SUBAPPLICATION LinksRechts_T_FF_Event (* Links/Rechts Umschaltung mittels Toggle-Flip-Flop (E_T_FF, Event/BOOL-basiert, keine Adapter). Schwester-Baustein zu MyLib::sys::AX_LinksRechts_T_FF (dort AX-Adapter-basiert). *)
  (* Standard: 61499-2 *)
  (* Version 1.0, 2026-09-09, Franz Höpfinger, Meisterschulen am Ostbahnhof, Ausgelagert aus Uebung_006a3_sub zur Wiederverwendung. *)
  PACKAGE MyLib::sys;
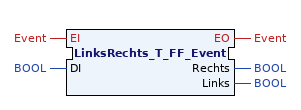
  EVENT_INPUT
    EI;
  END_EVENT
  EVENT_OUTPUT
    EO;
  END_EVENT
  VAR_INPUT
    DI : BOOL;
  END_VAR
  VAR_OUTPUT
    Rechts : BOOL;
    Links : BOOL;
  END_VAR
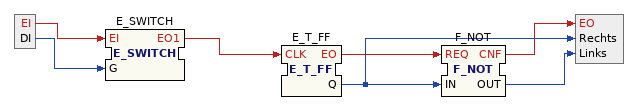
  FBS
    E_T_FF : iec61499::events::E_T_FF;
    E_SWITCH : iec61499::events::E_SWITCH;
    F_NOT : iec61131::bitwiseOperators::F_NOT;
  END_FBS
  EVENT_CONNECTIONS
    E_T_FF.EO TO F_NOT.REQ;
    EI TO E_SWITCH.EI;
    F_NOT.CNF TO EO;
    E_SWITCH.EO1 TO E_T_FF.CLK;
  END_CONNECTIONS
  DATA_CONNECTIONS
    E_T_FF.Q TO F_NOT.IN;
    E_T_FF.Q TO Rechts;
    DI TO E_SWITCH.G;
    F_NOT.OUT TO Links;
  END_CONNECTIONS
END_SUBAPPLICATION
